(* CoDeSys 2.3.9.45 project: CFC.pro *)
(* Libraries: Standard.lib 2.12.10 14:48:34, SYSLIBCALLBACK.LIB 2.12.10 14:48:32 *)

(* PLC configuration (modules and I/O channels)
K-Bus [K_Bus] node 0, in %IB0 out %QB0
Fieldbus variables [FB_VARS] node 1, in %IB0 out %QB0
Flag variables [FLAG_VARS] node 2, in %IB0 out %QB0
Modbus-Master [MB_MASTER] node 3, in %IB0 out %QB0
*)

(* POU PLC_PRG, CFC *)
PROGRAM PLC_PRG
VAR
END_VAR
VAR_INPUT
	S1: BOOL;
	S2: BOOL;
	S3: BOOL;
	S4: BOOL;
END_VAR

VAR_OUTPUT
	Q1: BOOL;
END_VAR
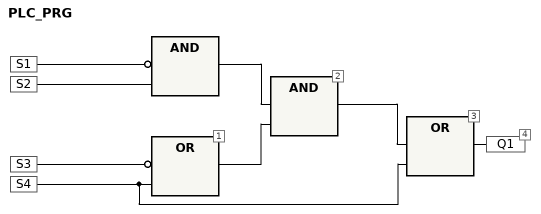
_CFC_ (* Continuous Function Chart, elements in execution order *)
#0 AND(NOT S1, S2)
#1 OR(NOT S3, S4)
#2 AND(#0, #1)
#3 OR(#2, S4)
#4 Q1 <= #3
_END_CFC_
(* the same logic as Structured Text *)
Q1 := ((NOT S1 AND S2) AND (NOT S3 OR S4)) OR S4;
END_PROGRAM
